# EPICS substitutions: IOC Files/hb2b-SE-Watlow_PM_IOC_Alarm.substitutions
file Watlow_PM_IOC_Alarms.template
{
pattern	{  s, ta,      ss}
		{HB2B, SE, Watlow}
}

file save_restoreStatus.db
{
pattern {P}
        {HB2B:CS:Watlow:}
}

file ioc_sns.db
{
pattern {IOCNAME}
        {HB2B:CS:Watlow}
}
